Fanuc TP program (LS listing): _clamp_down.ls

/PROG  _CLAMP_DOWN
/ATTR
OWNER		= MNEDITOR;
COMMENT		= "";
PROG_SIZE	= 229;
CREATE		= DATE 26-07-02  TIME 23:46:38;
MODIFIED	= DATE 26-07-02  TIME 23:46:38;
FILE_NAME	= _CLAMPDO;
VERSION		= 0;
LINE_COUNT	= 2;
MEMORY_SIZE	= 593;
PROTECT		= READ_WRITE;
TCD:  STACK_SIZE	= 0,
      TASK_PRIORITY	= 50,
      TIME_SLICE	= 0,
      BUSY_LAMP_OFF	= 0,
      ABORT_REQUEST	= 0,
      PAUSE_REQUEST	= 0;
DEFAULT_GROUP	= 1,*,*,*,*;
CONTROL_CODE	= 00000000 00000000;
LOCAL_REGISTERS	= 0,0,0;
/APPL

AUTO_SINGULARITY_HEADER;
  ENABLE_SINGULARITY_AVOIDANCE   : TRUE;
/MN
   1:  DO[66:OFF:Ret Clamp-Down]=ON ;
   2:  DO[65:OFF:Ext Clamp-Up]=OFF ;
/POS
/END
